TYPE E_AteqSequence :
(	
	IDLE, //DeviceIdle 
	PROGRAM_SELECT,
	RESET_FIFO,
	AUTO_ZERO,
	START_CYCLE, 
	LIVE_READING,
	END_OF_CYCLE,
	TIME_STAMP, 
	READ_LAST_RESULT,
	READ_FIFO,
	DONE
);
END_TYPE

(* stored: Version 1.1.0.1, ProductVersion 3.1.4024.15
   DUT E_AteqSequence: Id {e53874a6-2496-4372-b4ca-6316841d2cde} *)
